// TIA Portal V19 export
FUNCTION_BLOCK "Shutdown"   // FB12, LAD
{ S7_Optimized_Access := 'TRUE' }
// stored: AutoNumber false, MemoryReserve 100, SetENOAutomatically false
   VAR_INPUT
      shutdown : Bool;
   END_VAR
   VAR_OUTPUT
      returnValue : Word;
   END_VAR
   VAR
      statComment : String := 'Restart of Windows';
   END_VAR
BEGIN

REGION Network 1: Shutdown
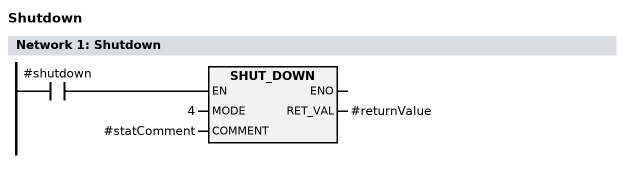
   RUNG wire#powerrail
      Contact( #shutdown )
      SHUT_DOWN(MODE := 4, COMMENT := #statComment, Ret_Val => #returnValue)
   END_RUNG
   // the same network as SCL:
   IF #shutdown THEN #returnValue := SHUT_DOWN(MODE := 4, COMMENT := #statComment); END_IF;
END_REGION
END_FUNCTION_BLOCK
